(* CoDeSys 2.3 export: TYPE.EXP *)

(* Data type *)
TYPE tAI :
STRUCT
	outVal:REAL;			(*Выходное значение*)
	TimeFiltr : TIME;		(*Время фильтрации*)
	n_Filtr : INT;			(*Количество данных для усреднения*)
	min_fiz : REAL;		(*Минимальное физическое значение*)
	max_fiz : REAL;		(*Максимальное физическое значение*)
	private : tSmoothParam;
END_STRUCT
END_TYPE

(* Data type *)
TYPE tDI :
STRUCT
	inVal:BOOL;
	outVal:BOOL;
	TimerDreb : TON;
	timeDreb:TIME;
	outVal_inv : BOOL;
END_STRUCT
END_TYPE

(* Data type *)
TYPE tDO :
STRUCT
	fActVal:BOOL;   	(*Активация*)
	fNewVal:BOOL;	(*Признак новой  команды*)
	fOldVal : BOOL;	(*Предыдущее значение*)
	fWriteVal:BOOL;	(*Записываемое значение*)
	fdefaultVal:BOOL;		(*Предустановленное значение*)
	fEnable:BOOL; 		(*Включение выхода*)
	ImpulseTimer:TON;	(*Таймер импульса*)

	TimeImp:TIME;

	TmrFlg		:BYTE;	(*ImpulseTimer,WaitInt,WaitPh*)


END_STRUCT
END_TYPE

(* Data type *)
TYPE tSmoothParam :
STRUCT
	b_Complete : BOOL; 	(*Флаг завершения фильтрации*)
	ind : INT;
	TimerFiltr : TON;		(*Таймер выборки значения при фильтрации*)
	arr_inputs : ARRAY [0..32] OF REAL;	(*,Буфер входных сигналов*)
	last_n : INT;
END_STRUCT
END_TYPE
